TYPE "LubrPump_Alr"
VERSION : 0.1
// Block: LubrPump_Alr
   STRUCT
      LowLevelLubrication : Bool;
   END_STRUCT;

END_TYPE
